Universal Robots PolyScope program: Gruppe6_16.03.urp

Program Gruppe6_16.03 (installation=default directory=/programs/usbdisk_0 createdIn=3.15.8.106339 lastSavedIn=3.15.8.106339 robotSerialNumber=2017355924)
Calibrated DH parameters: a=[0.000148, -0.262472, -0.392072, 0.000072, 0.000069, 0]; d=[0.089527, 96.545956, -95.500158, -0.935841, 0.094805, 0.082408]; alpha=[1.569624, 0.003467, 0.013158, 1.569531, -1.57018, 0]; deltaTheta=[-0.00002, 0.905644, -0.870628, -0.035105, 0.000064, 0.000046]
BeforeStart
  Set DigitalOutput pin=digital_out[1]; digitalValue=0
  Set DigitalOutput pin=config_out[0]; digitalValue=0
  MoveJ speed 60 deg/s, acceleration 80 deg/s^2 (useActiveTCP=true)
    Waypoint Waypoint_1: TCP in base x=199.763 y=-710.547 z=629.494 mm, rx=1.0347 ry=-0.9919 rz=2.1219 rad; joints [-65.96, -142.917, -12.798, 0.871, 92.276, -64.23] deg
Robot Program (runOnlyOnce=false)
  Wait Condition expression=config_out[0]≟ True
  Set DigitalOutput pin=config_out[0]; digitalValue=0
  Piece_x := read_port_register(128)/1000
  Piece_y := read_port_register(129)/-1000
  Piece_z := read_port_register(130)/1000
  Take_Piece := p[Piece_x,Piece_y,Piece_z,2.3,-2.2,0]
  Over_Piece := p[Piece_x,Piece_y,0.4,2.3,-2.2,0]
  MoveL speed 250 mm/s, acceleration 1200 mm/s^2 (useActiveTCP=true) feature=Base
    Waypoint Waypoint (Variable): variable=Over_Piece
    Waypoint Waypoint (Variable): variable=Take_Piece
    Set DigitalOutput pin=digital_out[1]; digitalValue=1
    Wait Condition expression=config_out[0]≟ True
    Set DigitalOutput pin=config_out[0]; digitalValue=0
    Set DigitalOutput pin=digital_out[1]; digitalValue=0
    Waypoint Waypoint (Variable): variable=Over_Piece
